(* IEC 61131-3 sources: programs/VI-54/VI-54_20171205/VI-54_20171205/Stations/PLC_VI54/VI-54_171014/Class/_LMC_MotorInfo, 1 file *)

(* ---- _LMC_MotorInfo.st ---- *)
(*!
<Class
	Name               = "_LMC_MotorInfo"
	Revision           = "6.1"
	RealtimeTask       = "false"
	CyclicTask         = "true"
	DefCyclictime      = "cCT"
	BackgroundTask     = "true"
	DefBackground      = "cBT"
	Sigmatek           = "false"
	OSInterface        = "false"
	HighPriority       = "false"
	Automatic          = "false"
	UpdateMode         = "Prescan"
	SharedCommandTable = "true"
	Objectsize         = "(870,1620)">
	<Channels>
		<Server Name="ActSpeed" Visualized="true" Initialize="false" WriteProtected="true" Retentive="false"/>
		<Server Name="AxleState" Visualized="true" Initialize="false" WriteProtected="true" Retentive="false"/>
		<Server Name="ClassSvr" Visualized="false" Initialize="false" WriteProtected="true" Retentive="false"/>
		<Server Name="CncOperationMode" Visualized="true" Initialize="false" WriteProtected="true" Retentive="false"/>
		<Server Name="DriveStateWord" Visualized="true" Initialize="false" WriteProtected="true" Retentive="false"/>
		<Server Name="Enabled" Visualized="true" Initialize="false" WriteProtected="true" Retentive="false"/>
		<Server Name="ExUnits" Visualized="true" Initialize="true" WriteProtected="false" Retentive="false"/>
		<Server Name="Homed" Visualized="true" Initialize="false" WriteProtected="true" Retentive="false"/>
		<Server Name="I_DERROR" Visualized="true" Initialize="false" WriteProtected="true" Retentive="false" Comment="Para-Nr : 201&#13;&#10;Unit  : [-]&#13;&#10;Description : Internal Drive Errors&#13;&#13;&#10;&#13;&#13;&#10;Bit 0 SSI_ERROR (additional Information to the Host Communication Error in [I-STATUS])&#13;&#10;Bit 1 HOST_ERROR (additional Information to the Host Communication Error in [I-STATUS])&#13;&#10;Bit 2 SHORT_ERROR (short of the power stage)&#13;&#10;Bit 3 RAM_ERROR (error in the code ram area)&#13;&#10;Bit 4 FPGA_WATCHDOG_ERROR &#13;&#10;Bit 5 ADOFF_ERROR (the offset of the motor current is to high)&#13;&#10;Bit 6 VCC18_ERROR (1,8V error)&#13;&#10;Bit 7 VCCE_ERROR (5V error)&#13;&#10;&#13;&#13;&#10;This bits cause the Drive Error Ramp/Drive Error No Ramp in [I-STATUS].&#13;&#13;&#10;Only bit 0 and 1 can be cleared by [K-CLRF].&#13;&#10;"/>
		<Server Name="I_I2T" Visualized="true" Initialize="false" WriteProtected="true" Retentive="false" Comment="Para-Nr : 193&#13;&#10;Unit  : [%]&#13;&#10;Description : Actual value of I2T of the power stage in % of [C-ICONT]&#13;&#13;&#10;&#13;&#13;&#10;The i2t-mechanism of the drive limits the current and the continuous current is always limited to the value of [C-ICONT].&#13;&#10;"/>
		<Server Name="I_ICMD" Visualized="true" Initialize="false" WriteProtected="true" Retentive="false" Comment="Para-Nr : 194&#13;&#10;Unit  : [mA]&#13;&#10;Description : Current set point in Q - direction"/>
		<Server Name="I_ICONT" Visualized="true" Initialize="false" WriteProtected="true" Retentive="false" Comment="Para-Nr : 186&#13;&#10;Unit  : [mA]&#13;&#10;Description : Drive continuos current&#13;&#10;"/>
		<Server Name="I_IPEAK" Visualized="true" Initialize="false" WriteProtected="true" Retentive="false" Comment="Para-Nr : 185&#13;&#10;Unit  : [mA]&#13;&#10;Description : Drive peak current&#13;&#10;"/>
		<Server Name="I_NCMD" Visualized="true" Initialize="false" WriteProtected="true" Retentive="false" Comment="Para-Nr : 190&#13;&#10;Unit  : [rpm]&#13;&#10;Description : Speed set point&#13;&#10;"/>
		<Server Name="I_PBAL" Visualized="true" Initialize="false" WriteProtected="true" Retentive="false" Comment="Para-Nr : 196&#13;&#10;Unit  : [W]&#13;&#10;Description : Actual regen power&#13;&#13;&#10;This value is influenced by [G-RBAL].&#13;&#10;"/>
		<Server Name="I_PE" Visualized="true" Initialize="false" WriteProtected="true" Retentive="false" Comment="Para-Nr : 175&#13;&#10;Unit  : [-]&#13;&#10;Description : Position error&#13;&#10;&#13;&#10;"/>
		<Server Name="I_STATUS" Visualized="true" Initialize="false" WriteProtected="true" Retentive="false" Comment="Para-Nr : 199&#13;&#10;Unit  : [-]&#13;&#10;Description : Status register:&#13;&#13;&#10;&#13;&#13;&#10;Bit  0   Mains phase (1-phase supply)&#13;&#10;Bit  1   Mains fault&#13;&#10;Bit  2   free (s e)&#13;&#10;Bit  3   Over voltage DC-Link&#13;&#10;Bit  4   Under voltage DC-link&#13;&#10;Bit  5   free (ad e)&#13;&#10;Bit  6   Holding brake error&#13;&#10;Bit  7   Holding brake switch damaged&#13;&#10;Bit  8   free&#13;&#10;Bit  9   Motor thermostat&#13;&#10;Bit 10  Ambient temperature&#13;&#10;Bit 11  Heat sink temperature&#13;&#10;Bit 12  Feedback Error&#13;&#10;Bit 13  Commutation error&#13;&#10;Bit 14  Over speed&#13;&#10;Bit 15  Contouring Error&#13;&#10;Bit 16  Trajectory Error&#13;&#10;Bit 17  Host Communication Error&#13;&#10;Bit 18  Drive Error Ramp, for additional information see [I-DERROR]&#13;&#10;Bit 19  Drive Error No Ramp, for additional information see [I-DERROR]&#13;&#10;Bit 20  External Enable Locked Error&#13;&#10;Bit 21  IGBT Driver Voltage Error&#13;&#10;Bit 22  max. Regen Power Error&#13;&#10;Bit 23  24V Brake Supply Error&#13;&#10;Bit 24  External Brake Enable Error&#13;&#10;Bit 25  I2T-Error&#13;&#10;Bit 26  Motor Temperature Warning&#13;&#10;&#13;&#13;&#10;The masks  [G-MASKE1], [G-MASKE2], [G-MASKW] and [G-MASKD] &#13;&#10;define if the corresponding bit of I-STATUS causes a cast of the motor, a ramp stop of the motor, a warning or nothing.&#13;&#13;&#10;This errors can be cleared with [K-CLRF].&#13;&#10;"/>
		<Server Name="I_TEMPE" Visualized="true" Initialize="false" WriteProtected="true" Retentive="false" Comment="Para-Nr : 184&#13;&#10;Unit  : [°C]&#13;&#10;Description : Actual ambient temperature&#13;&#10;"/>
		<Server Name="I_TEMPK" Visualized="true" Initialize="false" WriteProtected="true" Retentive="false" Comment="Para-Nr : 183&#13;&#10;Unit  : [°C]&#13;&#10;Description : Actual heat sink temperature&#13;&#10;&#13;&#10;"/>
		<Server Name="I_TEMPM" Visualized="true" Initialize="false" WriteProtected="true" Retentive="false" Comment="Para-Nr : 181&#13;&#10;Unit  : [Ohm]&#13;&#10;Description : Actual value of the PTC in the motor winding &#13;&#10;"/>
		<Server Name="I_VBUS" Visualized="true" Initialize="false" WriteProtected="true" Retentive="false" Comment="Para-Nr : 195&#13;&#10;Unit  : [V]&#13;&#10;Description : Actual DC-link voltage&#13;&#10;"/>
		<Server Name="IntUnits" Visualized="true" Initialize="true" WriteProtected="false" Retentive="false"/>
		<Server Name="MaxAccDec" Visualized="true" Initialize="true" WriteProtected="false" Retentive="false"/>
		<Server Name="MaxSpeed" Visualized="true" Initialize="true" WriteProtected="false" Retentive="false"/>
		<Server Name="Modulo" Visualized="true" Initialize="true" WriteProtected="false" Retentive="false"/>
		<Server Name="MoveType" Visualized="true" Initialize="true" WriteProtected="false" Retentive="false"/>
		<Server Name="SwMaxPos" Visualized="true" Initialize="true" WriteProtected="false" Retentive="false"/>
		<Server Name="SwMinPos" Visualized="true" Initialize="true" WriteProtected="false" Retentive="false"/>
		<Server Name="Tjerk" Visualized="true" Initialize="true" WriteProtected="false" Retentive="false"/>
		<Client Name="_DriveActValues1" Required="true" Internal="true"/>
		<Client Name="CNCState" Required="true" Internal="true"/>
		<Client Name="DriveAxis" Required="true" Internal="false" Comment="object channel to _DriveAxis"/>
		<Client Name="DriveStateW" Required="true" Internal="true"/>
		<Client Name="LMC" Required="true" Internal="false"/>
		<Client Name="LMC2" Required="false" Internal="false"/>
		<Client Name="LMC3" Required="false" Internal="false"/>
		<Client Name="SDDDriveError" Required="true" Internal="true"/>
		<Client Name="SDDDriveState" Required="true" Internal="true"/>
	</Channels>
	<Dependencies>
		<Files>
			<File Path=".\Class\_LMC_MotorInfo\_LMC_MotorInfo.vov"/>
		</Files>
	</Dependencies>
	<Network Name="_LMC_MotorInfo">
		<!-- List of Components in this network -->
		<Components>
			<Object
				Name       = "_DriveActValues1"
				Class      = "_DriveActValues"
				Position   = "(210,270)"
				Visualized = "true">
				<Channels>
					<Server Name="I_BCC"/>
					<Server Name="I_BITS"/>
					<Server Name="I_CAP"/>
					<Server Name="I_CAP4"/>
					<Server Name="I_CAPENC"/>
					<Server Name="I_DERROR"/>
					<Server Name="I_FBB"/>
					<Server Name="I_FPOS"/>
					<Server Name="I_I2T"/>
					<Server Name="I_IA"/>
					<Server Name="I_IB"/>
					<Server Name="I_ICMD"/>
					<Server Name="I_ICONT"/>
					<Server Name="I_ID"/>
					<Server Name="I_INT1"/>
					<Server Name="I_INT2"/>
					<Server Name="I_IPEAK"/>
					<Server Name="I_IQ"/>
					<Server Name="I_MPOS"/>
					<Server Name="I_N"/>
					<Server Name="I_NCMD"/>
					<Server Name="I_NFILT"/>
					<Server Name="I_PBAL"/>
					<Server Name="I_PCMD"/>
					<Server Name="I_PE"/>
					<Server Name="I_POS"/>
					<Server Name="I_STATUS"/>
					<Server Name="I_TEMPE"/>
					<Server Name="I_TEMPK"/>
					<Server Name="I_TEMPM"/>
					<Server Name="I_VBUS"/>
					<Server Name="State"/>
					<Client Name="DriveAxis"/>
					<Client Name="ErrorCode"/>
				</Channels>
			</Object>
			<Object
				Name       = "CNCState"
				Class      = "String"
				Position   = "(270,120)"
				Visualized = "true">
				<Channels>
					<Server Name="Data"/>
					<Client Name="SingleRealloc" Value="1"/>
				</Channels>
			</Object>
			<Object
				Name       = "DriveStateW"
				Class      = "String"
				Position   = "(300,2520)"
				Visualized = "true">
				<Channels>
					<Server Name="Data"/>
					<Client Name="SingleRealloc" Value="1"/>
				</Channels>
			</Object>
			<Object
				Name       = "SDDDriveError"
				Class      = "String"
				Position   = "(330,2400)"
				Visualized = "true">
				<Channels>
					<Server Name="Data"/>
					<Client Name="SingleRealloc" Value="1"/>
				</Channels>
			</Object>
			<Object
				Name       = "SDDDriveState"
				Class      = "String"
				Position   = "(300,2250)"
				Visualized = "true">
				<Channels>
					<Server Name="Data"/>
					<Client Name="SingleRealloc" Value="1"/>
				</Channels>
			</Object>
		</Components>
		<Comments>
		</Comments>
		<!-- List of Connections in this network -->
		<Connections>
			<Connection Source="this._DriveActValues1" Destination="_DriveActValues1.State"/>
			<Connection Source="_DriveActValues1.DriveAxis" Destination="this.DriveAxis" Vertices="(210,360),(38,210),"/>
			<Connection Source="this.I_PE" Destination="_DriveActValues1.I_PE" Vertices="(968,270),(796,480),"/>
			<Connection Source="this.I_TEMPM" Destination="_DriveActValues1.I_TEMPM" Vertices="(968,330),(796,720),"/>
			<Connection Source="this.I_TEMPK" Destination="_DriveActValues1.I_TEMPK" Vertices="(968,390),(796,780),"/>
			<Connection Source="this.I_TEMPE" Destination="_DriveActValues1.I_TEMPE" Vertices="(968,450),(796,840),"/>
			<Connection Source="this.I_IPEAK" Destination="_DriveActValues1.I_IPEAK" Vertices="(968,510),(796,900),"/>
			<Connection Source="this.I_ICONT" Destination="_DriveActValues1.I_ICONT" Vertices="(968,570),(796,960),"/>
			<Connection Source="this.I_NCMD" Destination="_DriveActValues1.I_NCMD" Vertices="(968,630),(796,1020),"/>
			<Connection Source="this.I_I2T" Destination="_DriveActValues1.I_I2T" Vertices="(968,690),(796,1200),"/>
			<Connection Source="this.I_ICMD" Destination="_DriveActValues1.I_ICMD" Vertices="(968,750),(796,1260),"/>
			<Connection Source="this.I_VBUS" Destination="_DriveActValues1.I_VBUS" Vertices="(968,810),(796,1320),"/>
			<Connection Source="this.CNCState" Destination="CNCState.Data"/>
			<Connection Source="this.I_STATUS" Destination="_DriveActValues1.I_STATUS" Vertices="(968,930),(796,1560),"/>
			<Connection Source="this.I_DERROR" Destination="_DriveActValues1.I_DERROR" Vertices="(968,990),(796,1620),"/>
			<Connection Source="this.SDDDriveState" Destination="SDDDriveState.Data"/>
			<Connection Source="this.SDDDriveError" Destination="SDDDriveError.Data"/>
			<Connection Source="this.DriveStateW" Destination="DriveStateW.Data"/>
			<Connection Source="this.I_PBAL" Destination="_DriveActValues1.I_PBAL" Vertices="(968,870),(796,1380),"/>
		</Connections>
		<!-- Headerfiles -->
		<Options>
		</Options>
	</Network>
</Class>
*)
_LMC_MotorInfo : CLASS
  //Servers:
	ClassSvr 	: SvrChCmd_DINT;
	I_PE 	: SvrCh_DINT;
	I_TEMPM 	: SvrCh_DINT;
	I_TEMPK 	: SvrCh_DINT;
	I_TEMPE 	: SvrCh_DINT;
	I_IPEAK 	: SvrCh_DINT;
	I_ICONT 	: SvrCh_DINT;
	I_NCMD 	: SvrCh_DINT;
	I_I2T 	: SvrCh_DINT;
	I_ICMD 	: SvrCh_DINT;
	I_VBUS 	: SvrCh_DINT;
	I_PBAL 	: SvrCh_DINT;
	I_STATUS 	: SvrCh__SDDISTATE;
	I_DERROR 	: SvrCh__SDDIDERROR;
	DriveStateWord 	: SvrCh_DS402_State;
	CncOperationMode 	: SvrCh__LMCAXIS_OPMODE;
	AxleState 	: SvrCh__LMCAXIS_STATUS;
	Enabled 	: SvrCh_DINT;
	Homed 	: SvrCh_DINT;
	ActSpeed 	: SvrCh_DINT;
	ExUnits 	: SvrCh_DINT;
	IntUnits 	: SvrCh_DINT;
	MaxSpeed 	: SvrCh_DINT;
	MaxAccDec 	: SvrCh_DINT;
	Tjerk 	: SvrCh_DINT;
	MoveType 	: SvrCh__LMCAXIS_MOVEPROFILE;
	Modulo 	: SvrCh_DINT;
	SwMinPos 	: SvrCh_DINT;
	SwMaxPos 	: SvrCh_DINT;
  //Clients:
	_DriveActValues1 	: CltChCmd__DriveActValues;
	DriveAxis 	: CltChCmd__DriveAxisBase;
	LMC 	: CltChCmd__LMCAxis;
	CNCState 	: CltChCmd_String;
	SDDDriveState 	: CltChCmd_String;
	SDDDriveError 	: CltChCmd_String;
	DriveStateW 	: CltChCmd_String;
	LMC2 	: CltChCmd__LMCAxis;
	LMC3 	: CltChCmd__LMCAxis;
  //Variables:
		BitNr 	: DINT;
		i 	: DINT;
		Lengte 	: UDINT;
		AxleStateTemp 	: _LMCAXIS_STATUS;
		DriveStateWordTemp 	: DS402_State;
		DriveI_status 	: _SDDISTATE;
		SDDDriveI_derror 	: _SDDIDERROR;
		AxleStateChar : ARRAY [0..31] OF CHAR;

		DriveStateChar : ARRAY [0..31] OF CHAR;

		SDDDriveStateChar : ARRAY [0..31] OF CHAR;

		SDDDriveErrorChar : ARRAY [0..31] OF CHAR;

		hSetValue 	: DINT;
		eenmaal 	: DINT;
		IndexFileNbr 	: DINT;
		OldExUnits 	: DINT;
		NewInterneUnits 	: DINT;
		NewMaxAccDec 	: DINT;
		NewMaxSpeed 	: DINT;
		CalcRatio 	: REAL;
		CalcMaxSpeed 	: DINT;
  //Functions:

	FUNCTION VIRTUAL GLOBAL Init;

	FUNCTION VIRTUAL GLOBAL CyWork
		VAR_INPUT
			EAX 	: UDINT;
		END_VAR
		VAR_OUTPUT
			state (EAX) 	: UDINT;
		END_VAR;

	FUNCTION VIRTUAL GLOBAL Background
		VAR_INPUT
			EAX 	: UDINT;
		END_VAR
		VAR_OUTPUT
			state (EAX) 	: UDINT;
		END_VAR;

	FUNCTION GLOBAL MyCyWork;

	FUNCTION GLOBAL MyBackGround;

	FUNCTION VIRTUAL GLOBAL I_PE::Read
		VAR_OUTPUT
			output (EAX) 	: DINT;
		END_VAR;

	FUNCTION VIRTUAL GLOBAL I_TEMPM::Read
		VAR_OUTPUT
			output (EAX) 	: DINT;
		END_VAR;

	FUNCTION VIRTUAL GLOBAL I_TEMPK::Read
		VAR_OUTPUT
			output (EAX) 	: DINT;
		END_VAR;

	FUNCTION VIRTUAL GLOBAL I_TEMPE::Read
		VAR_OUTPUT
			output (EAX) 	: DINT;
		END_VAR;

	FUNCTION VIRTUAL GLOBAL I_IPEAK::Read
		VAR_OUTPUT
			output (EAX) 	: DINT;
		END_VAR;

	FUNCTION VIRTUAL GLOBAL I_ICONT::Read
		VAR_OUTPUT
			output (EAX) 	: DINT;
		END_VAR;

	FUNCTION VIRTUAL GLOBAL I_NCMD::Read
		VAR_OUTPUT
			output (EAX) 	: DINT;
		END_VAR;

	FUNCTION VIRTUAL GLOBAL I_I2T::Read
		VAR_OUTPUT
			output (EAX) 	: DINT;
		END_VAR;

	FUNCTION VIRTUAL GLOBAL I_ICMD::Read
		VAR_OUTPUT
			output (EAX) 	: DINT;
		END_VAR;

	FUNCTION VIRTUAL GLOBAL I_VBUS::Read
		VAR_OUTPUT
			output (EAX) 	: DINT;
		END_VAR;

	FUNCTION VIRTUAL GLOBAL I_PBAL::Read
		VAR_OUTPUT
			output (EAX) 	: DINT;
		END_VAR;

	FUNCTION VIRTUAL GLOBAL I_STATUS::Read
		VAR_OUTPUT
			output (EAX) 	: _SDDISTATE;
		END_VAR;

	FUNCTION VIRTUAL GLOBAL I_DERROR::Read
		VAR_OUTPUT
			output (EAX) 	: _SDDIDERROR;
		END_VAR;
  //Tables:
	FUNCTION @STD
		VAR_OUTPUT
			ret_code	: CONFSTATES;
		END_VAR;
	FUNCTION GLOBAL TAB @CT_;
END_CLASS;

#pragma using _DriveActValues
#pragma using String
#pragma usingLtd _DriveAxisBase
#pragma usingLtd _LMCAxis

FUNCTION VIRTUAL GLOBAL _LMC_MotorInfo::Init

  _DriveActValues1.Init();

  if _FirstScan = 1 then
    eenmaal := 1;
  end_if;

END_FUNCTION

FUNCTION VIRTUAL GLOBAL _LMC_MotorInfo::CyWork
	VAR_INPUT
		EAX 	: UDINT;
	END_VAR
	VAR_OUTPUT
		state (EAX) 	: UDINT;
	END_VAR

  MyCyWork();

	state := READY;

END_FUNCTION

FUNCTION VIRTUAL GLOBAL _LMC_MotorInfo::Background
	VAR_INPUT
		EAX 	: UDINT;
	END_VAR
	VAR_OUTPUT
		state (EAX) 	: UDINT;
	END_VAR

  MyBackGround();

	state := READY;

END_FUNCTION

FUNCTION VIRTUAL GLOBAL _LMC_MotorInfo::I_PE::Read
	VAR_OUTPUT
		output (EAX) 	: DINT;
	END_VAR

	I_PE := _DriveActValues1.I_PE.Read();
	output := I_PE;

END_FUNCTION

FUNCTION VIRTUAL GLOBAL _LMC_MotorInfo::I_TEMPM::Read
	VAR_OUTPUT
		output (EAX) 	: DINT;
	END_VAR

	I_TEMPM := _DriveActValues1.I_TEMPM.Read();
	output := I_TEMPM;

END_FUNCTION

FUNCTION VIRTUAL GLOBAL _LMC_MotorInfo::I_TEMPK::Read
	VAR_OUTPUT
		output (EAX) 	: DINT;
	END_VAR

	I_TEMPK := _DriveActValues1.I_TEMPK.Read();
	output := I_TEMPK;

END_FUNCTION

FUNCTION VIRTUAL GLOBAL _LMC_MotorInfo::I_TEMPE::Read
	VAR_OUTPUT
		output (EAX) 	: DINT;
	END_VAR

	I_TEMPE := _DriveActValues1.I_TEMPE.Read();
	output := I_TEMPE;

END_FUNCTION

FUNCTION VIRTUAL GLOBAL _LMC_MotorInfo::I_IPEAK::Read
	VAR_OUTPUT
		output (EAX) 	: DINT;
	END_VAR

	I_IPEAK := _DriveActValues1.I_IPEAK.Read();
	output := I_IPEAK;

END_FUNCTION

FUNCTION VIRTUAL GLOBAL _LMC_MotorInfo::I_ICONT::Read
	VAR_OUTPUT
		output (EAX) 	: DINT;
	END_VAR

	I_ICONT := _DriveActValues1.I_ICONT.Read();
	output := I_ICONT;

END_FUNCTION

FUNCTION VIRTUAL GLOBAL _LMC_MotorInfo::I_NCMD::Read
	VAR_OUTPUT
		output (EAX) 	: DINT;
	END_VAR

	I_NCMD := _DriveActValues1.I_NCMD.Read();
	output := I_NCMD;

END_FUNCTION

FUNCTION VIRTUAL GLOBAL _LMC_MotorInfo::I_I2T::Read
	VAR_OUTPUT
		output (EAX) 	: DINT;
	END_VAR

	I_I2T := _DriveActValues1.I_I2T.Read() * 10;  // #pvo 141013  display waarde van xxx -> xxx.x
	output := I_I2T;

END_FUNCTION

FUNCTION VIRTUAL GLOBAL _LMC_MotorInfo::I_ICMD::Read
	VAR_OUTPUT
		output (EAX) 	: DINT;
	END_VAR

	I_ICMD := _DriveActValues1.I_ICMD.Read();
	output := I_ICMD;

END_FUNCTION

FUNCTION VIRTUAL GLOBAL _LMC_MotorInfo::I_VBUS::Read
	VAR_OUTPUT
		output (EAX) 	: DINT;
	END_VAR

	I_VBUS := _DriveActValues1.I_VBUS.Read();
	output := I_VBUS;

END_FUNCTION

FUNCTION VIRTUAL GLOBAL _LMC_MotorInfo::I_STATUS::Read
	VAR_OUTPUT
		output (EAX) 	: _SDDISTATE;
	END_VAR

	I_STATUS := _DriveActValues1.I_STATUS.Read();
	output := I_STATUS;

END_FUNCTION

FUNCTION VIRTUAL GLOBAL _LMC_MotorInfo::I_DERROR::Read
	VAR_OUTPUT
		output (EAX) 	: _SDDIDERROR;
	END_VAR

	I_DERROR := _DriveActValues1.I_DERROR.Read();
	output := I_DERROR;

END_FUNCTION

FUNCTION VIRTUAL GLOBAL _LMC_MotorInfo::I_PBAL::Read
	VAR_OUTPUT
		output (EAX) 	: DINT;
	END_VAR

	I_PBAL := _DriveActValues1.I_PBAL.Read();
	output := I_PBAL;

END_FUNCTION

FUNCTION GLOBAL _LMC_MotorInfo::MyCyWork

  _DriveActValues1.CyWork(EAX:=eax);
  DriveStateWord := DriveAxis.StateWord;

  LMC := LMC.Read();
  CncOperationMode := LMC;

  AxleState := LMC.ReadAxisStatus();
  ActSpeed := LMC.ReadVelocity(Mode:= LMCAXIS_SETVEL_APPUNIT_SEC);

END_FUNCTION

FUNCTION GLOBAL _LMC_MotorInfo::MyBackGround

// LMC axle state
  i := 32;
  AxleStateTemp := AxleState;
  while i > 0 do
    AxleStateChar[i-1] := (AxleStateTemp$usint AND 2#1 = 1);
    AxleStateChar[i-1] += '0';
    i -= 1;
    AxleStateTemp := AxleStateTemp SHR 1;
  end_while;
  Lengte := sizeof(AxleStateChar);
  CNCState.WriteDataOff(udLen:= Lengte, udOff:=0, pData:= #AxleStateChar$usint);

// SDDDrive State
  i := 32;
  DriveI_status := I_STATUS;
  while i > 0 do
    SDDDriveStateChar[i-1] := (DriveI_status$usint AND 2#1 = 1);
    SDDDriveStateChar[i-1] += '0';
    i -= 1;
    DriveI_status := DriveI_status SHR 1;
  end_while;
  Lengte := sizeof(SDDDriveStateChar);
  SDDDriveState.WriteDataOff(udLen:= Lengte, udOff:=0, pData:= #SDDDriveStateChar$usint);

// SDDDriveError
  i := 32;
  SDDDriveI_derror := I_DERROR;
  while i > 0 do
    SDDDriveErrorChar[i-1] := (SDDDriveI_derror$usint AND 2#1 = 1);
    SDDDriveErrorChar[i-1] += '0';
    i -= 1;
    SDDDriveI_derror := SDDDriveI_derror SHR 1;
  end_while;
  Lengte := sizeof(SDDDriveErrorChar);
  SDDDriveError.WriteDataOff(udLen:= Lengte, udOff:=0, pData:= #SDDDriveErrorChar$usint);

 // Drive State word
  i := 32;
  DriveStateWordTemp := DriveStateWord;
  while i > 0 do
    DriveStateChar[i-1] := (DriveStateWordTemp$usint AND 2#1 = 1);
    DriveStateChar[i-1] += '0';
    i -= 1;
    DriveStateWordTemp := DriveStateWordTemp SHR 1;
  end_while;
  Lengte := sizeof(DriveStateChar);
  DriveStateW.WriteDataOff(udLen:= Lengte, udOff:=0, pData:= #DriveStateChar$usint);

  Enabled := (AxleState.PowerOn = 1);
  Homed   := (AxleState.IsReferenced = 1);

  if eenmaal = 1 then
    // #pvo 150924
    LMC.ExUnits :=  ExUnits;
    LMC.ExUnits.Write(input:=ExUnits);

    LMC.IntUnits := IntUnits;
    LMC.IntUnits.Write(input:=IntUnits);

    LMC.VMax := MaxSpeed;
    LMC.VMax.Write(input:=MaxSpeed);

    LMC.AMax := MaxAccDec;
    LMC.AMax.Write(input:=MaxAccDec);

    LMC.Tjerk := Tjerk;
    LMC.Tjerk.Write(input:=Tjerk);

    LMC.MoveType := MoveType;
    LMC.MoveType.Write(input:=MoveType);

    LMC.SWMinPos := SwMinPos;
    LMC.SWMinPos.Write(input:=SwMinPos);

    LMC.SWMaxPos:= SwMaxPos;
    LMC.SWMaxPos.Write(input:=SwMaxPos);

    LMC.Modulo := Modulo;
    LMC.Modulo.Write(input:= Modulo);

    if IsClientConnected(#LMC2) then
    // #pvo 150924
      LMC2.ExUnits :=  ExUnits;
      LMC2.ExUnits.Write(input:=ExUnits);

      LMC2.IntUnits := IntUnits;
      LMC2.IntUnits.Write(input:=IntUnits);

      LMC2.VMax := MaxSpeed;
      LMC2.VMax.Write(input:=MaxSpeed);

      LMC2.AMax := MaxAccDec;
      LMC2.AMax.Write(input:=MaxAccDec);

      LMC2.Tjerk := Tjerk;
      LMC2.Tjerk.Write(input:=Tjerk);

      LMC2.MoveType := MoveType;
      LMC2.MoveType.Write(input:=MoveType);

      LMC2.SWMinPos := SwMinPos;
      LMC2.SWMinPos.Write(input:=SwMinPos);

      LMC2.SWMaxPos:= SwMaxPos;
      LMC2.SWMaxPos.Write(input:=SwMaxPos);

      LMC2.Modulo := Modulo;
      LMC2.Modulo.Write(input:= Modulo);
    end_if;

    if IsClientConnected(#LMC3) then
    // #pvo 150924
      LMC3.ExUnits :=  ExUnits;
      LMC3.ExUnits.Write(input:=ExUnits);

      LMC3.IntUnits := IntUnits;
      LMC3.IntUnits.Write(input:=IntUnits);

      LMC3.VMax := MaxSpeed;
      LMC3.VMax.Write(input:=MaxSpeed);

      LMC3.AMax := MaxAccDec;
      LMC3.AMax.Write(input:=MaxAccDec);

      LMC3.Tjerk := Tjerk;
      LMC3.Tjerk.Write(input:=Tjerk);

      LMC3.MoveType := MoveType;
      LMC3.MoveType.Write(input:=MoveType);

      LMC3.SWMinPos := SwMinPos;
      LMC3.SWMinPos.Write(input:=SwMinPos);

      LMC3.SWMaxPos:= SwMaxPos;
      LMC3.SWMaxPos.Write(input:=SwMaxPos);

      LMC3.Modulo := Modulo;
      LMC3.Modulo.Write(input:= Modulo);
    end_if;

     eenmaal := 0;
  end_if;

END_FUNCTION
